TEXTLIST MissionText
  0 = 'No Operation'
  1 = 'Init'
  2 = 'Picking...'
  3 = 'Picked'
  4 = 'Loading...'
  5 = 'Loaded'
  6 = 'Placing...'
  7 = 'Placed'
  8 = 'Unloading...'
  9 = 'Unloaded'
  10 = 'End'
  99 = 'Error'
   = ''
END_TEXTLIST

(* stored: Version 1.1.0.1, ProductVersion 3.1.4024.11
   TextList MissionText: Id {83ce7fd6-74c7-4c5f-a412-276d4870afc1} *)
